{attribute 'GeneratedUsingTerminal: KL8610-0002'}
{attribute addProperty BoxType "KL8610-0002"}
{attribute addProperty Id "KL8601_1AT %Q*KL_6576A6810KL8601_2AT %Q*KL_6576A6810KL8601_3AT %Q*KL_6576A6810"}
{attribute addProperty CRC "3209338988"}
{attribute addProperty Size "0"}
TYPE KL_BF4AA06C :
STRUCT
	{attribute addProperty Name "KL8601_1"}
	KL8601_1 : KL_6576A681;
	{attribute addProperty Name "KL8601_2"}
	KL8601_2 : KL_6576A681;
	{attribute addProperty Name "KL8601_3"}
	KL8601_3 : KL_6576A681;
END_STRUCT
END_TYPE

(* stored: Version 1.2.0.0, ProductVersion 3.1.4024.9
   DUT KL_BF4AA06C: Id {60e3f916-118c-4c11-834b-38af2faf8215} *)
